// TIA Portal V17 export
// export: Created 2024-10-17T14:16:18.0828858Z, ExportSetting WithDefaults, DisplayName Totally Integrated Automation Portal, DisplayVersion V17 Update 4, DisplayName TIA Portal Openness, DisplayVersion V17 Update 4, DisplayName TIA Portal Version Control Interface, DisplayVersion V17, DisplayName SINAMICS Startdrive Advanced, DisplayVersion V17 Update2, DisplayName SINAMICS Startdrive G130, G150, S120, S150, SINAMICS MV, S210, DisplayVersion V17 Update2, DisplayName SINAMICS Startdrive G110M, G120, G120C, G120D, G120P, G115D, DisplayVersion V17 Update2, DisplayName STEP 7 Professional, DisplayVersion V17 Update 4, DisplayName STEP 7 Safety, DisplayVersion V17, DisplayName WinCC Advanced / Unified PC, DisplayVersion V17 Update 4
TYPE "LPMLV2022_typeParameter_LREAL"
TITLE = LPMLV2022_typeParameter_LREAL
// Support: tech.team.motioncontrol@siemens.com
// stored: IsFailsafeCompliant false
   STRUCT
      ID : DInt;   // ID Value of Parameter. This is the arbitrary (user defined) ID value of the parameter
      "Name" : String[80];   // Name of Parameter. The literal parameter name is used to describe the parameter number, and its associated value
      Unit : String[6];   // Unit of Measure of Parameter. An example parameter unit of measure may be DegF, secs, PPM, revs, mm, etc.
      Value : LReal;   // Value of Parameter. This is the numeric value of the parameter
   END_STRUCT;
END_TYPE
